# EPICS substitutions: apps/mccApp/Db/hallb_ia.substitutions
file "db/hallb_ia_1.template" {
    pattern { P }
    { C1068_QDAC07 }
    { C1068_QDAC08 }
    { C1068_QDAC09 }
    { C1068_QDAC10 }
}
